// TwinCAT 3 PLC project PLC_Sim
// ProgramVersion: 3.1.4024.0
// libraries:
//   Tc2_Standard, * (Beckhoff Automation GmbH)
//   Tc2_System, * (Beckhoff Automation GmbH)
//   Tc3_Module, * (Beckhoff Automation GmbH)
//   VisuDialogs, * (System)
//   VisuSymbols,3.5.10.0,System
// project tree:
//   / GlobalTextList.TcGTLO, PlcTask.TcTTO, Visualization Manager.TcVMO (not stored)
//   GVLs/ GVL.TcGVL
//   POUs/ Example.TcPOU, MAIN.TcPOU, Reset.TcPOU, V0_1.TcPOU, V0_10.TcPOU, V0_11.TcPOU, V0_2.TcPOU, V0_3.TcPOU, V0_4.TcPOU, V0_5.TcPOU, V0_6.TcPOU, V0_7.TcPOU, V0_8.TcPOU, V0_9.TcPOU
//   VISUs/ Visualization.TcVIS
// real-time tasks:
//   TASK PlcTask: cycle T#10ms, priority 20, ADS port 350
// I/O:
//   DEVICE Device 1 (EtherCAT) (disabled), AmsNetId 10.181.16.108.2.1
//     Term 1 (EK1200) [EK1200-5000 EtherCAT Power supply (2A E-Bus)]
//       Term 2 (EL1008) [EL1008 8Ch. Dig. Input 24V, 3ms]
//       Term 3 (EL2008) [EL2008 8Ch. Dig. Output 24V, 0.5A]
//       Term 4 (EL2008) [EL2008 8Ch. Dig. Output 24V, 0.5A]
//       Term 5 (EL4001) [EL4001 1Ch. Ana. Output 0-10V, 12bit]
//       Term 6 (EL3062) [EL3062 2Ch. Ana. Input 0-10V]
//       Term 7 (EL9011) [EL9011 End Terminal]
//   DEVICE Device 3 (NOV-DP-RAM) (disabled)
// variable links:
//   PLC_Sim/PLC_Sim Instance <-> Device 1 (EtherCAT)/Term 1 (EK1200)/Term 2 (EL1008)
//     PlcTask Inputs/MAIN.bButton_1_PLC <-> Channel 1/Input
//   PLC_Sim/PLC_Sim Instance <-> Device 1 (EtherCAT)/Term 1 (EK1200)/Term 3 (EL2008)
//     PlcTask Outputs/MAIN.bLamp_1_PLC <-> Channel 1/Output

CONFIGURATION PLC_Sim
    RESOURCE PLC ON TwinCAT3
        TASK PlcTask(INTERVAL := T#10ms, PRIORITY := 20);
        PROGRAM MAIN WITH PlcTask : MAIN;
    END_RESOURCE
END_CONFIGURATION

// ---- GVLs/GVL.TcGVL
{attribute 'qualified_only'}
VAR_GLOBAL
	// Inputs
	// Buttons
	bButton_1 : BOOL;
	bButton_2 : BOOL;
	bButton_3 : BOOL;
	bButton_4 : BOOL;
	bButton_5 : BOOL;
	bButton_6 : BOOL;
	bButton_7 : BOOL;
	bButton_8 : BOOL;
	// Switches
	bSwitch_1 : BOOL;
	bSwitch_2 : BOOL;
	bSwitch_3 : BOOL;
	bSwitch_4 : BOOL;
	bSwitch_5 : BOOL;
	bSwitch_6 : BOOL;
	bSwitch_7 : BOOL;
	bSwitch_8 : BOOL;
	// Potentiometer
	fPotentiometer_1 : REAL;
	fPotentiometer_2 : REAL;
	
	// Outputs
	// Lamps
	bLamp_1 : BOOL;
	bLamp_2 : BOOL;
	bLamp_3 : BOOL;
	bLamp_4 : BOOL;
	bLamp_5 : BOOL;
	bLamp_6 : BOOL;
	bLamp_7 : BOOL;
	bLamp_8 : BOOL;
	// Meter
	fMeter_1 : REAL;
	fMeter_2 : REAL;
	
	// Running program ID
	nProgramID : UINT := 0;
	
	// I/O Setting
	bUsePLC : bool := false;
END_VAR

// ---- POUs/MAIN.TcPOU
PROGRAM MAIN
VAR
	nPreviusProgramID : UINT := 0;
	
	// Link to PLC (Optional)
	bButton_1_PLC AT %I* : BOOL;
	bButton_2_PLC AT %I* : BOOL;
	bButton_3_PLC AT %I* : BOOL;
	bButton_4_PLC AT %I* : BOOL;
	
	bLamp_1_PLC AT %Q* : BOOL;
	bLamp_2_PLC AT %Q* : BOOL;
	bLamp_3_PLC AT %Q* : BOOL;
	bLamp_4_PLC AT %Q* : BOOL;
END_VAR

// Auto Reset VISU
IF nPreviusProgramID <> GVL.nProgramID THEN
	nPreviusProgramID := GVL.nProgramID;
	Reset();
END_IF

// PLC Link
IF GVL.bUsePLC THEN
	GVL.bButton_1 := bButton_1_PLC;
	GVL.bButton_2 := bButton_2_PLC;
	GVL.bButton_3 := bButton_3_PLC;
	GVL.bButton_4 := bButton_4_PLC;
	
	bLamp_1_PLC := GVL.bLamp_1;
	bLamp_2_PLC := GVL.bLamp_2;
	bLamp_3_PLC := GVL.bLamp_3;
	bLamp_4_PLC := GVL.bLamp_4;
END_IF;

// Program List
CASE GVL.nProgramID OF
	0 : Reset();
	1 : V0_1();
	2 : V0_2();
	3 : V0_3();
	4 : V0_4();
	5 : V0_5();
	6 : V0_6();
	7 : V0_7();
	8 : V0_8();
	9 : V0_9();
	10 : V0_10();
	11 : V0_11();
END_CASE

END_PROGRAM

// ---- POUs/Reset.TcPOU
PROGRAM Reset
VAR
END_VAR

// Inputs
// Buttons
GVL.bButton_1 := FALSE;
GVL.bButton_2 := FALSE;
GVL.bButton_3 := FALSE;
GVL.bButton_4 := FALSE;
GVL.bButton_5 := FALSE;
GVL.bButton_6 := FALSE;
GVL.bButton_7 := FALSE;
GVL.bButton_8 := FALSE;
// Switches
GVL.bSwitch_1 := FALSE;
GVL.bSwitch_2 := FALSE;
GVL.bSwitch_3 := FALSE;
GVL.bSwitch_4 := FALSE;
GVL.bSwitch_5 := FALSE;
GVL.bSwitch_6 := FALSE;
GVL.bSwitch_7 := FALSE;
GVL.bSwitch_8 := FALSE;
// Potentiometer
GVL.fPotentiometer_1 := 0;
GVL.fPotentiometer_2 := 0;

// Outputs
// Lamps
GVL.bLamp_1 := FALSE;
GVL.bLamp_2 := FALSE;
GVL.bLamp_3 := FALSE;
GVL.bLamp_4 := FALSE;
GVL.bLamp_5 := FALSE;
GVL.bLamp_6 := FALSE;
GVL.bLamp_7 := FALSE;
GVL.bLamp_8 := FALSE;
// Meter
GVL.fMeter_1 := 0;
GVL.fMeter_2 := 0;

// Running program ID
//GVL.nProgramID := 0;

END_PROGRAM

// ---- POUs/V0_1.TcPOU
PROGRAM V0_1
VAR
END_VAR

(*
	Ja-functie
	
	Het meest eenvoudige dat men kan programmeren is de JA-functie. Bij de JA-functie volgt de uitgang de ingang.
	Als de ingang logisch '1' is, is de uitgang logisch '1'. Als de ingang logisch '0' is, is de uitgang logisch '0'.
*)

GVL.bLamp_1 := GVL.bButton_1;

END_PROGRAM

// ---- POUs/V0_2.TcPOU
PROGRAM V0_2
VAR
END_VAR

(*
	Twee signalen
	
	Als S01=1 en S02=0 moet Q01 branden
	Als S01=0 en S02=1 moet Q02 branden
	Als S01=0 en S02=0 moet Q01 en Q02 branden
	Als S01=1 en S02=1 moet Q01 en Q02 niet branden
	
	S1	S2	Q1	Q2
	0	0	1	1
	0	1	0	1
	1	0	1	0
	1	1	0	0
*)

GVL.bLamp_1 := (NOT GVL.bSwitch_2);
GVL.bLamp_2 := (NOT GVL.bSwitch_1);

END_PROGRAM

// ---- POUs/V0_3.TcPOU
PROGRAM V0_3
VAR
END_VAR

(*
	Reactorvat
	
	De installatie zal pas werken als een hoofdschakelaar S01 AAN staat (maakcontact).
	Als het niveau in het vat te hoog is, reageert detector S03.
	Als de temperatuur boven een bepaalde waarde stijgt reageert thermostaat S04.
	Als de druk boven een bepaalde waarde stijgt reageert druksensor S05.
	Als één van de drie detectoren (S03, S04, S05) reageert moet een oranje lamp Q01 branden.
	Als twee van de drie detectoren reageert moet een rode lamp Q02 branden.
	Als de detectoren alle drie reageren moeten beide lampen branden en ook een bel Q03 rinkelen.
	De bel blijft rinkelen tot de stopdrukknop S02 ingedrukt wordt (verbreekcontact).
	
	S1	S3	S4	S5	Q1	Q2	Q3
	0	x	x	x	0	0	0
	
	1	1	0	0	1	0	0
	1	0	1	0	1	0	0
	1	0	0	1	1	0	0
	
	1	1	1	0	1	1	0
	1	0	1	1	1	1	0
	1	1	0	1	1	1	0
	
	1	1	1	1	1	1	1
*)

GVL.bLamp_1 := GVL.bSwitch_1 AND (GVL.bSwitch_2 OR GVL.bSwitch_3 OR GVL.bSwitch_4);
GVL.bLamp_2 := GVL.bSwitch_1 AND ((GVL.bSwitch_2 AND GVL.bSwitch_3) OR (GVL.bSwitch_2 AND GVL.bSwitch_4) OR (GVL.bSwitch_3 AND GVL.bSwitch_4));
GVL.bLamp_3 := GVL.bSwitch_1 AND GVL.bSwitch_2 AND GVL.bSwitch_3 AND GVL.bSwitch_4;

END_PROGRAM

// ---- POUs/V0_4.TcPOU
PROGRAM V0_4
VAR
END_VAR

(*
	Opslagvat
	
	Een opslagvat heeft twee sensoren in de zijwand die een laag en hoog niveau aanduiden. Aan de hand van een PLC programma dient er
	automatisch de klep bovenaan het vat geopend te worden als het vat leeg is. De tank wordt nu gevuld. Als de tank vol is
	sluit de klep K1 eveneens automatisch. Onderaan de tank bevindt zich een pomp P1 die met een start- en stop-drukknop in- en
	uitgeschakeld kan worden. 

	Als de tank leeg gelopen is, stopt de pomp automatisch en opent de klep K1 bovenaan. De pomp kan niet ingeschakeld worden
	zolang de tank gevuld wordt.
	
	(T = Toggle)
	L1	l2	S1	P1	K1
	0	0	x	x	1
	1	0	x	x	1
	1	1	x	x	0
	
	x	x	0	0T	x
	x	x	1	1T	x
*)

GVL.bLamp_1 := NOT GVL.bSwitch_1; // L2

GVL.bLamp_2 R= (GVL.bButton_1 AND GVL.bLamp_2) OR (NOT GVL.bSwitch_1);
GVL.bLamp_2 S= GVL.bButton_2 AND NOT GVL.bLamp_2 AND GVL.bSwitch_1;

END_PROGRAM

// ---- POUs/V0_5.TcPOU
PROGRAM V0_5
VAR
END_VAR

(*
	Opslagvat met foutdetectie
	
	In de voorgaande oefening werden twee sensoren voor niveaudetectie gebruikt. Het is onmogelijk dat de sensor onderaan geen vloeistof detecteert (FALSE)
	en de sensor bovenaan de tank wel (TRUE). De sensor onderaan moet dus defect zijn of er is een kabelbreuk. In dat geval mogen noch de klep, noch de pomp geactiveerd kunnen worden.
	
	bSwitch_1 = Hoog niveau (L1)
	bSwitch_2 = Laag niveau (L2)
	bLamp_1 = Klep (K1)
	bLamp_2 = Pomp (P1)
	bButton_1 = Pomp start (B1)
	bButton_2 = Pomp stop (B2)
	
	(T = Toggle)
	L1	l2	B1	B2	P1	K1
	0	0	x	x	x	1	-- Sturing klep
	1	0	x	x	x	0
	1	1	x	x	x	0
	0	1	x	x	x	1
	
	x	1	1	0	1	x	-- Sturing pomp
	x	1	0	1	0	x
	x	0	x	x	0	x	
*)

// Sturing klep
GVL.bLamp_1 := (NOT GVL.bSwitch_1 AND NOT GVL.bSwitch_2) OR (NOT GVL.bSwitch_1 AND GVL.bSwitch_2);

// Sturing pomp
GVL.bLamp_2 S= GVL.bSwitch_2 AND GVL.bButton_1;
GVL.bLamp_2 R= (GVL.bSwitch_2 AND GVL.bButton_2) OR (GVL.bSwitch_1 AND NOT GVL.bSwitch_2) OR NOT GVL.bSwitch_2;

END_PROGRAM

// ---- POUs/V0_6.TcPOU
PROGRAM V0_6
VAR
END_VAR

(*
	Alarmbewaking
	
	In een vat wordt een proces bewaakt met 3 sensoren:
    	Sensor1 meet de druk. TRUE bij een te hoge druk.
    	Sensor2 meet de temperatuur. TRUE bij een te hoge temperatuur.
    	Sensor3 meet het vloeistofniveau. FALSE bij een te laag niveau.

	Er zijn 5 lampen die als indicator dienen voor het proces:
    	Lamp1 gaat aan als de druk te hoog is.
    	Lamp2 gaat aan als de temperatuur te hoog is.
    	Lamp3 gaat aan als het niveau te laag is.
    		Bovenstaande lampen gaan automatisch uit als er geen melding meer gegeven hoeft te worden.
    	Lamp4 gaat aan als er zich twee alarmen gelijktijdig voordoen. Van zodra er geen twee alarmen meer zijn gaat deze lamp uit. Bij drie alarmen gaat deze lamp ook uit.
    	Lamp5 gaat aan als er drie alarmen zijn. Deze lamp blijft aan, ook nadat er geen drie alarmen meer zijn. De lamp kan enkel uitgeschakeld worden met een extra drukknop.
	
	bSwitch_1 = Sensor 1 (S1)
	bSwitch_2 = Sensor 2 (S2)
	bSwitch_3 = Sensor 3 (S3)
	bButton_1 = Drukknop (B1) -- Reset voor 3 alarmen
	
	bLamp_1 = Lemp 1 (L1)
	bLamp_2 = Lamp 2 (L2)
	bLamp_3 = Lamp 3 (L3)
	bLamp_4 = Lamp 4 (L4)
	bLamp_5 = Lamp 5 (L5)
	
	(T = Toggle)
	S1	S2	S3	B1		L1	L2	L3	L4	L5
	1	x	x	x		1	x	x	x	x
	x	1	x	x		x	1	x	x	x
	x	x	0	x		x	x	1	x	x
	
	0	1	1	x		x	x	x	1	x	-- Andere zijn uit
	1	0	1	x		x	x	x	1	x
	1	1	0	x		x	x	x	1	x
	
	1	1	1	x		x	x	x	x	1T
	x	x	x	1		x	x	x	x	0T
*)

GVL.bLamp_1 := GVL.bSwitch_1;
GVL.bLamp_2 := GVL.bSwitch_2;
GVL.bLamp_3 := NOT GVL.bSwitch_3;

GVL.bLamp_4 := ((GVL.bSwitch_1 AND GVL.bSwitch_2) OR (GVL.bSwitch_1 AND NOT GVL.bSwitch_3) OR (GVL.bSwitch_2 AND NOT GVL.bSwitch_3)) AND NOT (GVL.bSwitch_1 AND GVL.bSwitch_2 AND NOT GVL.bSwitch_3);

GVL.bLamp_5 S= GVL.bSwitch_1 AND GVL.bSwitch_2 AND NOT GVL.bSwitch_3;
GVL.bLamp_5 R= GVL.bLamp_5 AND GVL.bButton_1 AND NOT (GVL.bSwitch_1 AND GVL.bSwitch_2 AND NOT GVL.bSwitch_3);

END_PROGRAM

// ---- POUs/V0_7.TcPOU
PROGRAM V0_7
VAR
	bOn : BOOL;
	bOff : BOOL;
END_VAR
(*
	Teleruptorschakeling | uitleg
	
	In woningen wordt een soortgelijke schakeling gebruikt om de verlichting in en uit te schakelen door gebruik te maken van parallel geschakelde drukknoppen. Men noemt het ook soms een afstands- of trappenhuisschakelaar. Maak deze na in LADDER en probeer te achterhalen hoe deze werkt.

	Zorg ervoor dat er meerdere drukknoppen (op ieder verdiep) gebruikt kunnen worden.

	De P in het maakcontact Ingang zorgt ervoor dat deze puls- of flank-gestuurd is. Deze kan je eenvoudig toevoegen door het maakcontact te selecteren en de P-toets op je toetsenbord in te drukken.

	De tussenvariable M0 wordt in de PLC wereld een Merker genoemd. Deze is nodig omdat je in LADDER een maakcontact niet kan inverteren alsook flankgestuurd maken.

	Je zal wel gemerkt hebben dat in het tweede netwerk de NO maakcontact lamp parallel met NO maakcontact M0 als een overneemcontact werkt. De NC merker M0 en NC lamp die omgekeerd in serie staan zorgen ervoor dat dit onderbroken kan worden
*)
VAR // added by the converter: edge detectors and wires of the graphical bodies
    _rt1, _rt2, _rt3, _rt4 : R_TRIG;
END_VAR

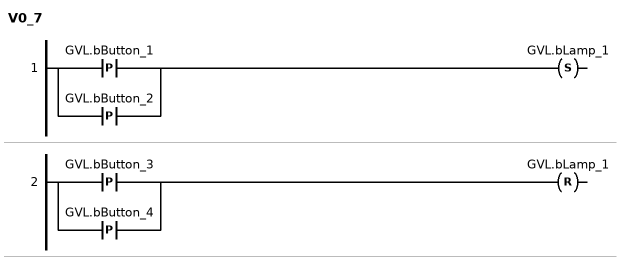
// NETWORK 1
_rt1(CLK := GVL.bButton_1);
_rt2(CLK := GVL.bButton_2);
GVL.bLamp_1 S= _rt1.Q OR _rt2.Q;

// NETWORK 2
_rt3(CLK := GVL.bButton_3);
_rt4(CLK := GVL.bButton_4);
GVL.bLamp_1 R= _rt3.Q OR _rt4.Q;

END_PROGRAM

// ---- POUs/V0_8.TcPOU
PROGRAM V0_8
VAR
	fbOn : R_TRIG;
	fbOff : R_TRIG;
	
	bOnTrigger : BOOL;
	bOffTrigger : BOOL;
END_VAR

(*
	Teleruptorschakeling
	
	Programmeer de teleruptorschakeling in Structured Tekst. Zorg ook hier dat het mogelijk is om te bedienen met meerdere drukknoppen. Je zal merken dat dit een veel eenvoudiger programma zal zijn dan in LADDER. 

	Voor de flank-detectie heb je een Function Block (FB) nodig. Met een rechtermuisklik in het programmeervenster (niet het declareer venster) kan de 'input assisant' openen en selecteer vervolgens > Function Blocks > Tc2_Standard > trigger > R_TRIG
*)

fbOn(CLK := GVL.bButton_1 OR GVL.bButton_2, Q => bOnTrigger);
fbOff(CLK := GVL.bButton_3 OR GVL.bButton_4, Q => bOffTrigger);

GVL.bLamp_1 S= bOnTrigger;
GVL.bLamp_1 R= bOffTrigger;

END_PROGRAM

// ---- POUs/V0_9.TcPOU
PROGRAM V0_9
VAR
	fbRTrig : R_TRIG;
	bTrigger : BOOL;
	nState : SINT := 0;
END_VAR

(*
	Motor starten met één drukknop
	
	Schrijf een programma om een motor [ Relais voor MotorLinks en MotorRechts ] te starten en te stoppen met één drukknop. De installatie zal pas werken als een hoofdschakelaar AAN staat.
		1e druk op de drukknop:	start links draaiend
		2e druk op de drukknop:	stop
		3e druk op de drukknop:	start rechts draaiend
		4e druk op de drukknop:	stop
	
	bSwitch_1 = Hoofdschakelaar
	bButton_1 = Drukknop
	bLamp_1 = Links om
	bLamp_2 = Rechts om
*)

fbRTrig(CLK := GVL.bButton_1, Q => bTrigger);

END_PROGRAM

// ---- POUs/V0_10.TcPOU
PROGRAM V0_10
VAR
END_VAR

(*
	Twee Pompen
	
	Een tank wordt gevuld met twee pompen. Om onderhoud te vermijden en de slijtage aan de pompen te spreiden zal men elke pomp om beurten apart laten werken. De installatie zal pas werken als een hoofdschakelaar AAN staat.

	De pompbeweging wordt gestart ofwel:
    	manueel door een startdrukknop
    	automatisch door een niveauschakelaar (onderin de tank)

	De pompbeweging wordt gestopt ofwel:
    	manueel door een stopdrukknop
    	automatisch door een niveauschakelaar (bovenaan de tank)
*)

END_PROGRAM

// ---- POUs/V0_11.TcPOU
PROGRAM V0_11
VAR
END_VAR

(*
	Drie pompen
	
	Een tank wordt gevuld met drie pompen. De installatie zal pas werken als een hoofdschakelaar AAN staat. Om het debiet te regelen kunnen achtereenvolgens één, twee of alle drie
	de pompen tegelijk worden ingeschakeld. Dit gebeurt met één enkele drukknop. Een andere drukknop zal op elk moment alle pompen uitschakelen.
*)

END_PROGRAM

// ---- POUs/Example.TcPOU
PROGRAM Example
VAR
END_VAR

GVL.bLamp_1 := GVL.bButton_1 AND GVL.bSwitch_1;
GVL.bLamp_2 := GVL.bButton_2 AND NOT GVL.bSwitch_2;
GVL.bLamp_3 := GVL.bButton_3 OR GVL.bSwitch_3;
GVL.bLamp_4 := GVL.bButton_4 OR NOT GVL.bSwitch_4;
GVL.bLamp_5 := GVL.bButton_5 OR GVL.bSwitch_5;
GVL.bLamp_6 := GVL.bButton_6 OR GVL.bSwitch_6;
GVL.bLamp_7 := GVL.bButton_7 OR GVL.bSwitch_7;
GVL.bLamp_8 := GVL.bButton_8 OR GVL.bSwitch_8;

GVL.fMeter_1 := GVL.fPotentiometer_1 * 1200 / 10 - 200; // -200 - 1000 range
GVL.fMeter_2 := GVL.fPotentiometer_2 * 100 / 10; // 0 - 100 range

END_PROGRAM

// ---- GlobalTextList.TcGTLO
TEXTLIST GlobalTextList
  67 = ''
  815 = '%f'
  893 = '%i'
  463 = 'BTN 1'
  613 = 'BTN 2'
  100 = 'BTN 3'
  691 = 'BTN 4'
  166 = 'Button 1'
  10 = 'Button 2'
  299 = 'Button 3'
  673 = 'Button 4'
  503 = 'Button 5'
  408 = 'Button 6'
  211 = 'Button 7'
  308 = 'Button 8'
  890 = 'Click to change'
  692 = 'Click to change running program'
  502 = 'Enable PLC Output'
  374 = 'Lamp 1'
  340 = 'Lamp 2'
  569 = 'Lamp 3'
  461 = 'Lamp 4'
  663 = 'Lamp 5'
  662 = 'Lamp 6'
  462 = 'Lamp 7'
  530 = 'Lamp 8'
  276 = 'Running program:'
  766 = 'Switch 1'
  987 = 'Switch 2'
  81 = 'Switch 3'
  521 = 'Switch 4'
  697 = 'Switch 5'
  667 = 'Switch 6'
  911 = 'Switch 7'
  672 = 'Switch 8'
  19 = 'test'
  173 = 'Toggles between PLC I/O or VISU I/O'
  810 = 'Visualization created by Lenny Industries'
END_TEXTLIST

// ---- VISUs/Visualization.TcVIS
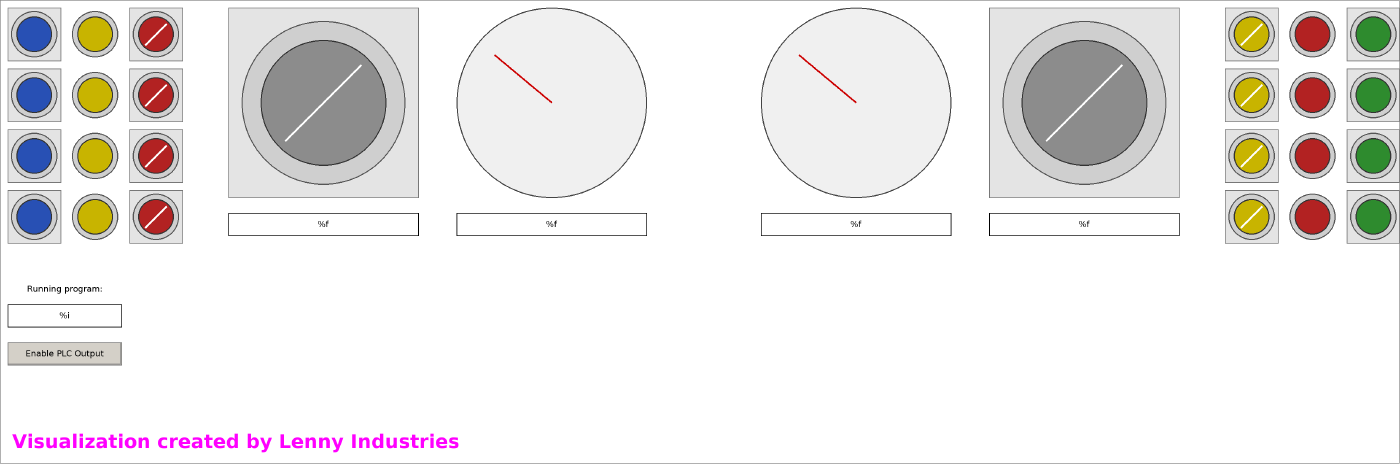
VISUALIZATION Visualization  // 1840x610
    PushSwitch (10,10 70x70), tooltip "Button 1", variable: GVL.bButton_1, behaviour: TAP, style: Switch-PushSwitch-Blue
    PushSwitch (10,90 70x70), tooltip "Button 2", variable: GVL.bButton_2, behaviour: TAP, style: Switch-PushSwitch-Blue
    PushSwitch (10,170 70x70), tooltip "Button 3", variable: GVL.bButton_3, behaviour: TAP, style: Switch-PushSwitch-Blue
    PushSwitch (10,250 70x70), tooltip "Button 4", variable: GVL.bButton_4, behaviour: TAP, style: Switch-PushSwitch-Blue
    Lamp1 (90,10 70x70), tooltip "Lamp 1", variable: GVL.bLamp_1, style: Lamp-Lamp1-Yellow
    Lamp1 (90,90 70x70), tooltip "Lamp 2", variable: GVL.bLamp_2, style: Lamp-Lamp1-Yellow
    Lamp1 (90,170 70x70), tooltip "Lamp 3", variable: GVL.bLamp_3, style: Lamp-Lamp1-Yellow
    Lamp1 (90,250 70x70), tooltip "Lamp 4", variable: GVL.bLamp_4, style: Lamp-Lamp1-Yellow
    RotarySwitch (170,10 70x70), tooltip "Switch 1", variable: GVL.bSwitch_1, behaviour: TOGGLE, style: Switch-RotarySwitch-Red
    RotarySwitch (170,90 70x70), tooltip "Switch 2", variable: GVL.bSwitch_2, behaviour: TOGGLE, style: Switch-RotarySwitch-Red
    RotarySwitch (170,170 70x70), tooltip "Switch 3", variable: GVL.bSwitch_3, behaviour: TOGGLE, style: Switch-RotarySwitch-Red
    RotarySwitch (170,250 70x70), tooltip "Switch 4", variable: GVL.bSwitch_4, behaviour: TOGGLE, style: Switch-RotarySwitch-Red
    Meter360 (600,10 250x250), value: GVL.fMeter_1, style: Meter-Meter360-Gray, scale format: %.1f, scale -200..1000
    Potentiometer360 (300,10 250x250), variable: GVL.fPotentiometer_1, style: Potentiometer-Potentiometer360-Gray, scale format: %.1f, scale 0..10
    Rectangle (300,280 250x30), "%f", tooltip "Click to change", text variable: GVL.fPotentiometer_1
        OnMouseDown: write the text variable via VisuDialogs.Numpad, min 0, max 10, format %f
    Rectangle (600,280 250x30), "%f", text variable: GVL.fMeter_1
    Label (10,550 600x60), "Visualization created by Lenny Industries"
    Meter360 (1000,10 250x250), value: GVL.fMeter_2, style: Meter-Meter360-Gray, scale format: %.1f, scale 0..100
    Potentiometer360 (1300,10 250x250), variable: GVL.fPotentiometer_2, style: Potentiometer-Potentiometer360-Gray, scale format: %.1f, scale 0..10
    Rectangle (1300,280 250x30), "%f", tooltip "Click to change", text variable: GVL.fPotentiometer_2
        OnMouseDown: write the text variable via VisuDialogs.Numpad, min 0, max 10, format %f
    Rectangle (1000,280 250x30), "%f", text variable: GVL.fMeter_2
    PushSwitch (1770,10 70x70), tooltip "Button 5", variable: GVL.bButton_5, behaviour: TAP, style: Switch-PushSwitch-Green
    PushSwitch (1770,90 70x70), tooltip "Button 6", variable: GVL.bButton_6, behaviour: TAP, style: Switch-PushSwitch-Green
    PushSwitch (1770,170 70x70), tooltip "Button 7", variable: GVL.bButton_7, behaviour: TAP, style: Switch-PushSwitch-Green
    PushSwitch (1770,250 70x70), tooltip "Button 8", variable: GVL.bButton_8, behaviour: TAP, style: Switch-PushSwitch-Green
    Lamp1 (1690,10 70x70), tooltip "Lamp 5", variable: GVL.bLamp_5, style: Lamp-Lamp1-Red
    Lamp1 (1690,90 70x70), tooltip "Lamp 6", variable: GVL.bLamp_6, style: Lamp-Lamp1-Red
    Lamp1 (1690,170 70x70), tooltip "Lamp 7", variable: GVL.bLamp_7, style: Lamp-Lamp1-Red
    Lamp1 (1690,250 70x70), tooltip "Lamp 8", variable: GVL.bLamp_8, style: Lamp-Lamp1-Red
    RotarySwitch (1610,10 70x70), tooltip "Switch 5", variable: GVL.bSwitch_5, behaviour: TOGGLE, style: Switch-RotarySwitch-Yellow
    RotarySwitch (1610,90 70x70), tooltip "Switch 6", variable: GVL.bSwitch_6, behaviour: TOGGLE, style: Switch-RotarySwitch-Yellow
    RotarySwitch (1610,170 70x70), tooltip "Switch 7", variable: GVL.bSwitch_7, behaviour: TOGGLE, style: Switch-RotarySwitch-Yellow
    RotarySwitch (1610,250 70x70), tooltip "Switch 8", variable: GVL.bSwitch_8, behaviour: TOGGLE, style: Switch-RotarySwitch-Yellow
    Rectangle (10,400 150x30), "%i", tooltip "Click to change running program", text variable: GVL.nProgramID
        OnMouseDown: write the text variable via VisuDialogs.Numpad, min 0, max 65536, format %i
    Label (10,365 150x30), "Running program:"
    Button (10,450 150x30), "Enable PLC Output", tooltip "Toggles between PLC I/O or VISU I/O", colour toggle: GVL.bUsePLC
        toggle GVL.bUsePLC
END_VISUALIZATION
